	UF : 1, UT : 1,		CONFIG : 'N U T, 0, 0, 1',
	X =  103.000  mm,	Y =  238.000  mm,	Z =   15.000 mm,
	W =180.000 deg,	P =   0.000 deg,	R =    90.000 deg
};
P[11494]{
   GP1:
	UF : 1, UT : 1,		CONFIG : 'N U T, 0, 0, 1',
	X =  106.000  mm,	Y =  238.000  mm,	Z =   15.000 mm,
	W =180.000 deg,	P =   0.000 deg,	R =    90.000 deg
};
P[11495]{
   GP1:
	UF : 1, UT : 1,		CONFIG : 'N U T, 0, 0, 1',
	X =  106.000  mm,	Y =  238.000  mm,	Z =   0.600 mm,
	W =180.000 deg,	P =   0.000 deg,	R =    90.000 deg
};
P[11496]{
   GP1:
	UF : 1, UT : 1,		CONFIG : 'N U T, 0, 0, 1',
	X =  106.000  mm,	Y =  238.000  mm,	Z =   15.000 mm,
	W =180.000 deg,	P =   0.000 deg,	R =    90.000 deg
};
P[11497]{
   GP1:
	UF : 1, UT : 1,		CONFIG : 'N U T, 0, 0, 1',
	X =  109.000  mm,	Y =  238.000  mm,	Z =   15.000 mm,
	W =180.000 deg,	P =   0.000 deg,	R =    90.000 deg
};
P[11498]{
   GP1:
	UF : 1, UT : 1,		CONFIG : 'N U T, 0, 0, 1',
	X =  109.000  mm,	Y =  238.000  mm,	Z =   0.600 mm,
	W =180.000 deg,	P =   0.000 deg,	R =    90.000 deg
};
P[11499]{
   GP1:
	UF : 1, UT : 1,		CONFIG : 'N U T, 0, 0, 1',
	X =  109.000  mm,	Y =  238.000  mm,	Z =   15.000 mm,
	W =180.000 deg,	P =   0.000 deg,	R =    90.000 deg
};
P[11500]{
   GP1:
	UF : 1, UT : 1,		CONFIG : 'N U T, 0, 0, 1',
	X =  112.000  mm,	Y =  238.000  mm,	Z =   15.000 mm,
	W =180.000 deg,	P =   0.000 deg,	R =    90.000 deg
};
P[11501]{
   GP1:
	UF : 1, UT : 1,		CONFIG : 'N U T, 0, 0, 1',
	X =  112.000  mm,	Y =  238.000  mm,	Z =   0.600 mm,
	W =180.000 deg,	P =   0.000 deg,	R =    90.000 deg
};
P[11502]{
   GP1:
	UF : 1, UT : 1,		CONFIG : 'N U T, 0, 0, 1',
	X =  112.000  mm,	Y =  238.000  mm,	Z =   15.000 mm,
	W =180.000 deg,	P =   0.000 deg,	R =    90.000 deg
};
P[11503]{
   GP1:
	UF : 1, UT : 1,		CONFIG : 'N U T, 0, 0, 1',
	X =  115.000  mm,	Y =  238.000  mm,	Z =   15.000 mm,
	W =180.000 deg,	P =   0.000 deg,	R =    90.000 deg
};
P[11504]{
   GP1:
	UF : 1, UT : 1,		CONFIG : 'N U T, 0, 0, 1',
	X =  115.000  mm,	Y =  238.000  mm,	Z =   0.600 mm,
	W =180.000 deg,	P =   0.000 deg,	R =    90.000 deg
};
P[11505]{
   GP1:
	UF : 1, UT : 1,		CONFIG : 'N U T, 0, 0, 1',
	X =  115.000  mm,	Y =  238.000  mm,	Z =   15.000 mm,
	W =180.000 deg,	P =   0.000 deg,	R =    90.000 deg
};
P[11506]{
   GP1:
	UF : 1, UT : 1,		CONFIG : 'N U T, 0, 0, 1',
	X =  118.000  mm,	Y =  238.000  mm,	Z =   15.000 mm,
	W =180.000 deg,	P =   0.000 deg,	R =    90.000 deg
};
P[11507]{
   GP1:
	UF : 1, UT : 1,		CONFIG : 'N U T, 0, 0, 1',
	X =  118.000  mm,	Y =  238.000  mm,	Z =   0.600 mm,
	W =180.000 deg,	P =   0.000 deg,	R =    90.000 deg
};
P[11508]{
   GP1:
	UF : 1, UT : 1,		CONFIG : 'N U T, 0, 0, 1',
	X =  118.000  mm,	Y =  238.000  mm,	Z =   15.000 mm,
	W =180.000 deg,	P =   0.000 deg,	R =    90.000 deg
};
P[11509]{
   GP1:
	UF : 1, UT : 1,		CONFIG : 'N U T, 0, 0, 1',
	X =  121.000  mm,	Y =  238.000  mm,	Z =   15.000 mm,
	W =180.000 deg,	P =   0.000 deg,	R =    90.000 deg
};
P[11510]{
   GP1:
	UF : 1, UT : 1,		CONFIG : 'N U T, 0, 0, 1',
	X =  121.000  mm,	Y =  238.000  mm,	Z =   0.600 mm,
	W =180.000 deg,	P =   0.000 deg,	R =    90.000 deg
};
P[11511]{
   GP1:
	UF : 1, UT : 1,		CONFIG : 'N U T, 0, 0, 1',
	X =  121.000  mm,	Y =  238.000  mm,	Z =   15.000 mm,
	W =180.000 deg,	P =   0.000 deg,	R =    90.000 deg
};
P[11512]{
   GP1:
	UF : 1, UT : 1,		CONFIG : 'N U T, 0, 0, 1',
	X =  124.000  mm,	Y =  238.000  mm,	Z =   15.000 mm,
	W =180.000 deg,	P =   0.000 deg,	R =    90.000 deg
};
P[11513]{
   GP1:
	UF : 1, UT : 1,		CONFIG : 'N U T, 0, 0, 1',
	X =  124.000  mm,	Y =  238.000  mm,	Z =   0.600 mm,
	W =180.000 deg,	P =   0.000 deg,	R =    90.000 deg
};
P[11514]{
   GP1:
	UF : 1, UT : 1,		CONFIG : 'N U T, 0, 0, 1',
	X =  124.000  mm,	Y =  238.000  mm,	Z =   15.000 mm,
	W =180.000 deg,	P =   0.000 deg,	R =    90.000 deg
};
P[11515]{
   GP1:
	UF : 1, UT : 1,		CONFIG : 'N U T, 0, 0, 1',
	X =  127.000  mm,	Y =  238.000  mm,	Z =   15.000 mm,
	W =180.000 deg,	P =   0.000 deg,	R =    90.000 deg
};
P[11516]{
   GP1:
	UF : 1, UT : 1,		CONFIG : 'N U T, 0, 0, 1',
	X =  127.000  mm,	Y =  238.000  mm,	Z =   0.600 mm,
	W =180.000 deg,	P =   0.000 deg,	R =    90.000 deg
};
P[11517]{
   GP1:
	UF : 1, UT : 1,		CONFIG : 'N U T, 0, 0, 1',
	X =  127.000  mm,	Y =  238.000  mm,	Z =   15.000 mm,
	W =180.000 deg,	P =   0.000 deg,	R =    90.000 deg
};
P[11518]{
   GP1:
	UF : 1, UT : 1,		CONFIG : 'N U T, 0, 0, 1',
	X =  130.000  mm,	Y =  238.000  mm,	Z =   15.000 mm,
	W =180.000 deg,	P =   0.000 deg,	R =    90.000 deg
};
P[11519]{
   GP1:
	UF : 1, UT : 1,		CONFIG : 'N U T, 0, 0, 1',
	X =  130.000  mm,	Y =  238.000  mm,	Z =   0.600 mm,
	W =180.000 deg,	P =   0.000 deg,	R =    90.000 deg
};
P[11520]{
   GP1:
	UF : 1, UT : 1,		CONFIG : 'N U T, 0, 0, 1',
	X =  130.000  mm,	Y =  238.000  mm,	Z =   15.000 mm,
	W =180.000 deg,	P =   0.000 deg,	R =    90.000 deg
};
P[11521]{
   GP1:
	UF : 1, UT : 1,		CONFIG : 'N U T, 0, 0, 1',
	X =  133.000  mm,	Y =  238.000  mm,	Z =   15.000 mm,
	W =180.000 deg,	P =   0.000 deg,	R =    90.000 deg
};
P[11522]{
   GP1:
	UF : 1, UT : 1,		CONFIG : 'N U T, 0, 0, 1',
	X =  133.000  mm,	Y =  238.000  mm,	Z =   0.600 mm,
	W =180.000 deg,	P =   0.000 deg,	R =    90.000 deg
};
P[11523]{
   GP1:
	UF : 1, UT : 1,		CONFIG : 'N U T, 0, 0, 1',
	X =  133.000  mm,	Y =  238.000  mm,	Z =   15.000 mm,
	W =180.000 deg,	P =   0.000 deg,	R =    90.000 deg
};
P[11524]{
   GP1:
	UF : 1, UT : 1,		CONFIG : 'N U T, 0, 0, 1',
	X =  136.000  mm,	Y =  238.000  mm,	Z =   15.000 mm,
	W =180.000 deg,	P =   0.000 deg,	R =    90.000 deg
};
P[11525]{
   GP1:
	UF : 1, UT : 1,		CONFIG : 'N U T, 0, 0, 1',
	X =  136.000  mm,	Y =  238.000  mm,	Z =   0.600 mm,
	W =180.000 deg,	P =   0.000 deg,	R =    90.000 deg
};
P[11526]{
   GP1:
	UF : 1, UT : 1,		CONFIG : 'N U T, 0, 0, 1',
	X =  136.000  mm,	Y =  238.000  mm,	Z =   15.000 mm,
	W =180.000 deg,	P =   0.000 deg,	R =    90.000 deg
};
P[11527]{
   GP1:
	UF : 1, UT : 1,		CONFIG : 'N U T, 0, 0, 1',
	X =  139.000  mm,	Y =  238.000  mm,	Z =   15.000 mm,
	W =180.000 deg,	P =   0.000 deg,	R =    90.000 deg
};
P[11528]{
   GP1:
	UF : 1, UT : 1,		CONFIG : 'N U T, 0, 0, 1',
	X =  139.000  mm,	Y =  238.000  mm,	Z =   0.600 mm,
	W =180.000 deg,	P =   0.000 deg,	R =    90.000 deg
};
P[11529]{
   GP1:
	UF : 1, UT : 1,		CONFIG : 'N U T, 0, 0, 1',
	X =  139.000  mm,	Y =  238.000  mm,	Z =   15.000 mm,
	W =180.000 deg,	P =   0.000 deg,	R =    90.000 deg
};
P[11530]{
   GP1:
	UF : 1, UT : 1,		CONFIG : 'N U T, 0, 0, 1',
	X =  142.000  mm,	Y =  238.000  mm,	Z =   15.000 mm,
	W =180.000 deg,	P =   0.000 deg,	R =    90.000 deg
};
P[11531]{
   GP1:
	UF : 1, UT : 1,		CONFIG : 'N U T, 0, 0, 1',
	X =  142.000  mm,	Y =  238.000  mm,	Z =   0.600 mm,
	W =180.000 deg,	P =   0.000 deg,	R =    90.000 deg
};
P[11532]{
   GP1:
	UF : 1, UT : 1,		CONFIG : 'N U T, 0, 0, 1',
	X =  142.000  mm,	Y =  238.000  mm,	Z =   15.000 mm,
	W =180.000 deg,	P =   0.000 deg,	R =    90.000 deg
};
P[11533]{
   GP1:
	UF : 1, UT : 1,		CONFIG : 'N U T, 0, 0, 1',
	X =  145.000  mm,	Y =  238.000  mm,	Z =   15.000 mm,
	W =180.000 deg,	P =   0.000 deg,	R =    90.000 deg
};
P[11534]{
   GP1:
	UF : 1, UT : 1,		CONFIG : 'N U T, 0, 0, 1',
	X =  145.000  mm,	Y =  238.000  mm,	Z =   0.600 mm,
	W =180.000 deg,	P =   0.000 deg,	R =    90.000 deg
};
P[11535]{
   GP1:
	UF : 1, UT : 1,		CONFIG : 'N U T, 0, 0, 1',
	X =  145.000  mm,	Y =  238.000  mm,	Z =   15.000 mm,
	W =180.000 deg,	P =   0.000 deg,	R =    90.000 deg
};
P[11536]{
   GP1:
	UF : 1, UT : 1,		CONFIG : 'N U T, 0, 0, 1',
	X =  148.000  mm,	Y =  238.000  mm,	Z =   15.000 mm,
	W =180.000 deg,	P =   0.000 deg,	R =    90.000 deg
};
P[11537]{
   GP1:
	UF : 1, UT : 1,		CONFIG : 'N U T, 0, 0, 1',
	X =  148.000  mm,	Y =  238.000  mm,	Z =   0.600 mm,
	W =180.000 deg,	P =   0.000 deg,	R =    90.000 deg
};
P[11538]{
   GP1:
	UF : 1, UT : 1,		CONFIG : 'N U T, 0, 0, 1',
	X =  148.000  mm,	Y =  238.000  mm,	Z =   15.000 mm,
	W =180.000 deg,	P =   0.000 deg,	R =    90.000 deg
};
P[11539]{
   GP1:
	UF : 1, UT : 1,		CONFIG : 'N U T, 0, 0, 1',
	X =  151.000  mm,	Y =  238.000  mm,	Z =   15.000 mm,
	W =180.000 deg,	P =   0.000 deg,	R =    90.000 deg
};
P[11540]{
   GP1:
	UF : 1, UT : 1,		CONFIG : 'N U T, 0, 0, 1',
	X =  151.000  mm,	Y =  238.000  mm,	Z =   0.600 mm,
	W =180.000 deg,	P =   0.000 deg,	R =    90.000 deg
};
P[11541]{
   GP1:
	UF : 1, UT : 1,		CONFIG : 'N U T, 0, 0, 1',
	X =  151.000  mm,	Y =  238.000  mm,	Z =   15.000 mm,
	W =180.000 deg,	P =   0.000 deg,	R =    90.000 deg
};
P[11542]{
   GP1:
	UF : 1, UT : 1,		CONFIG : 'N U T, 0, 0, 1',
	X =  154.000  mm,	Y =  238.000  mm,	Z =   15.000 mm,
	W =180.000 deg,	P =   0.000 deg,	R =    90.000 deg
};
P[11543]{
   GP1:
	UF : 1, UT : 1,		CONFIG : 'N U T, 0, 0, 1',
	X =  154.000  mm,	Y =  238.000  mm,	Z =   0.600 mm,
	W =180.000 deg,	P =   0.000 deg,	R =    90.000 deg
};
P[11544]{
   GP1:
	UF : 1, UT : 1,		CONFIG : 'N U T, 0, 0, 1',
	X =  154.000  mm,	Y =  238.000  mm,	Z =   15.000 mm,
	W =180.000 deg,	P =   0.000 deg,	R =    90.000 deg
};
P[11545]{
   GP1:
	UF : 1, UT : 1,		CONFIG : 'N U T, 0, 0, 1',
	X =  157.000  mm,	Y =  238.000  mm,	Z =   15.000 mm,
	W =180.000 deg,	P =   0.000 deg,	R =    90.000 deg
};
P[11546]{
   GP1:
	UF : 1, UT : 1,		CONFIG : 'N U T, 0, 0, 1',
	X =  157.000  mm,	Y =  238.000  mm,	Z =   0.600 mm,
	W =180.000 deg,	P =   0.000 deg,	R =    90.000 deg
};
P[11547]{
   GP1:
	UF : 1, UT : 1,		CONFIG : 'N U T, 0, 0, 1',
	X =  157.000  mm,	Y =  238.000  mm,	Z =   15.000 mm,
	W =180.000 deg,	P =   0.000 deg,	R =    90.000 deg
};
P[11548]{
   GP1:
	UF : 1, UT : 1,		CONFIG : 'N U T, 0, 0, 1',
	X =  160.000  mm,	Y =  238.000  mm,	Z =   15.000 mm,
	W =180.000 deg,	P =   0.000 deg,	R =    90.000 deg
};
P[11549]{
   GP1:
	UF : 1, UT : 1,		CONFIG : 'N U T, 0, 0, 1',
	X =  160.000  mm,	Y =  238.000  mm,	Z =   0.600 mm,
	W =180.000 deg,	P =   0.000 deg,	R =    90.000 deg
};
P[11550]{
   GP1:
	UF : 1, UT : 1,		CONFIG : 'N U T, 0, 0, 1',
	X =  160.000  mm,	Y =  238.000  mm,	Z =   15.000 mm,
	W =180.000 deg,	P =   0.000 deg,	R =    90.000 deg
};
P[11551]{
   GP1:
	UF : 1, UT : 1,		CONFIG : 'N U T, 0, 0, 1',
	X =  163.000  mm,	Y =  238.000  mm,	Z =   15.000 mm,
	W =180.000 deg,	P =   0.000 deg,	R =    90.000 deg
};
P[11552]{
   GP1:
	UF : 1, UT : 1,		CONFIG : 'N U T, 0, 0, 1',
	X =  163.000  mm,	Y =  238.000  mm,	Z =   0.600 mm,
	W =180.000 deg,	P =   0.000 deg,	R =    90.000 deg
};
P[11553]{
   GP1:
	UF : 1, UT : 1,		CONFIG : 'N U T, 0, 0, 1',
	X =  163.000  mm,	Y =  238.000  mm,	Z =   15.000 mm,
	W =180.000 deg,	P =   0.000 deg,	R =    90.000 deg
};
P[11554]{
   GP1:
	UF : 1, UT : 1,		CONFIG : 'N U T, 0, 0, 1',
	X =  166.000  mm,	Y =  238.000  mm,	Z =   15.000 mm,
	W =180.000 deg,	P =   0.000 deg,	R =    90.000 deg
};
P[11555]{
   GP1:
	UF : 1, UT : 1,		CONFIG : 'N U T, 0, 0, 1',
	X =  166.000  mm,	Y =  238.000  mm,	Z =   0.600 mm,
	W =180.000 deg,	P =   0.000 deg,	R =    90.000 deg
};
P[11556]{
   GP1:
	UF : 1, UT : 1,		CONFIG : 'N U T, 0, 0, 1',
	X =  166.000  mm,	Y =  238.000  mm,	Z =   15.000 mm,
	W =180.000 deg,	P =   0.000 deg,	R =    90.000 deg
};
P[11557]{
   GP1:
	UF : 1, UT : 1,		CONFIG : 'N U T, 0, 0, 1',
	X =  169.000  mm,	Y =  238.000  mm,	Z =   15.000 mm,
	W =180.000 deg,	P =   0.000 deg,	R =    90.000 deg
};
P[11558]{
   GP1:
	UF : 1, UT : 1,		CONFIG : 'N U T, 0, 0, 1',
	X =  169.000  mm,	Y =  238.000  mm,	Z =   0.600 mm,
	W =180.000 deg,	P =   0.000 deg,	R =    90.000 deg
};
P[11559]{
   GP1:
	UF : 1, UT : 1,		CONFIG : 'N U T, 0, 0, 1',
	X =  169.000  mm,	Y =  238.000  mm,	Z =   15.000 mm,
	W =180.000 deg,	P =   0.000 deg,	R =    90.000 deg
};
P[11560]{
   GP1:
	UF : 1, UT : 1,		CONFIG : 'N U T, 0, 0, 1',
	X =  172.000  mm,	Y =  238.000  mm,	Z =   15.000 mm,
	W =180.000 deg,	P =   0.000 deg,	R =    90.000 deg
};
P[11561]{
   GP1:
	UF : 1, UT : 1,		CONFIG : 'N U T, 0, 0, 1',
	X =  172.000  mm,	Y =  238.000  mm,	Z =   0.600 mm,
	W =180.000 deg,	P =   0.000 deg,	R =    90.000 deg
};
P[11562]{
   GP1:
	UF : 1, UT : 1,		CONFIG : 'N U T, 0, 0, 1',
	X =  172.000  mm,	Y =  238.000  mm,	Z =   15.000 mm,
	W =180.000 deg,	P =   0.000 deg,	R =    90.000 deg
};
P[11563]{
   GP1:
	UF : 1, UT : 1,		CONFIG : 'N U T, 0, 0, 1',
	X =  175.000  mm,	Y =  238.000  mm,	Z =   15.000 mm,
	W =180.000 deg,	P =   0.000 deg,	R =    90.000 deg
};
P[11564]{
   GP1:
	UF : 1, UT : 1,		CONFIG : 'N U T, 0, 0, 1',
	X =  175.000  mm,	Y =  238.000  mm,	Z =   0.600 mm,
	W =180.000 deg,	P =   0.000 deg,	R =    90.000 deg
};
P[11565]{
   GP1:
	UF : 1, UT : 1,		CONFIG : 'N U T, 0, 0, 1',
	X =  175.000  mm,	Y =  238.000  mm,	Z =   15.000 mm,
	W =180.000 deg,	P =   0.000 deg,	R =    90.000 deg
};
P[11566]{
   GP1:
	UF : 1, UT : 1,		CONFIG : 'N U T, 0, 0, 1',
	X =  178.000  mm,	Y =  238.000  mm,	Z =   15.000 mm,
	W =180.000 deg,	P =   0.000 deg,	R =    90.000 deg
};
P[11567]{
   GP1:
	UF : 1, UT : 1,		CONFIG : 'N U T, 0, 0, 1',
	X =  178.000  mm,	Y =  238.000  mm,	Z =   0.600 mm,
	W =180.000 deg,	P =   0.000 deg,	R =    90.000 deg
};
P[11568]{
   GP1:
	UF : 1, UT : 1,		CONFIG : 'N U T, 0, 0, 1',
	X =  178.000  mm,	Y =  238.000  mm,	Z =   15.000 mm,
	W =180.000 deg,	P =   0.000 deg,	R =    90.000 deg
};
P[11569]{
   GP1:
	UF : 1, UT : 1,		CONFIG : 'N U T, 0, 0, 1',
	X =  145.000  mm,	Y =  300.000  mm,	Z =   150.000 mm,
	W =180.000 deg,	P =   0.000 deg,	R =    90.000 deg
};
/END
